SUBAPPLICATION Uebung_213c (* Standard IEC 61131-3 FB_CTU_UDINT (Vorwärtszähler, UDINT) mit Terminal-Ausgabe (PHYS_LREAL) *)
  (* Standard: 61131-3; Description: Copyright (c) 2026 Meisterschulen am Ostbahnhof This program and the accompanying materials are made available under the terms of the Eclipse Public License 2.0 which is available at https://www.eclipse.org/legal/epl-2.0/ SPDX-License-Identifier: EPL-2.0 *)
  (* Version 1.1, 2026-04-21, Franz Höpfinger, Meisterschulen am Ostbahnhof, Added terminal output for counter value (PHYS_LREAL, direct connection) *)
  (* Version 1.0, 2026-04-20, Franz Höpfinger, Meisterschulen am Ostbahnhof, initial API and implementation (IEC 61131-3 version) *)
  PACKAGE Uebungen;
  IMPORT Uebungen::const::UT::Horse::DefaultPool_Horse::Container_Horse;
  IMPORT Uebungen::const::UT::Horse::DefaultPool_Horse::ObjectPointer_Horse;
  IMPORT Uebungen::const::UT::Horse::DefaultPool_Horse::frame_00;
  IMPORT Uebungen::const::UT::Horse::DefaultPool_Horse::frame_01;
  IMPORT Uebungen::const::UT::Horse::DefaultPool_Horse::frame_02;
  IMPORT Uebungen::const::UT::Horse::DefaultPool_Horse::frame_03;
  IMPORT Uebungen::const::UT::Horse::DefaultPool_Horse::frame_04;
  IMPORT Uebungen::const::UT::Horse::DefaultPool_Horse::frame_05;
  IMPORT Uebungen::const::UT::Horse::DefaultPool_Horse::frame_06;
  IMPORT Uebungen::const::UT::Horse::DefaultPool_Horse::frame_07;
  IMPORT Uebungen::const::UT::Horse::DefaultPool_Horse::frame_08;
  IMPORT Uebungen::const::UT::Horse::DefaultPool_Horse::frame_09;
  IMPORT Uebungen::const::UT::Horse::DefaultPool_Horse::frame_10;
  IMPORT Uebungen::const::UT::Horse::DefaultPool_Horse::frame_11;
  IMPORT Uebungen::const::UT::Horse::DefaultPool_Horse::frame_12;
  IMPORT Uebungen::const::UT::Horse::DefaultPool_Horse::frame_13;
  IMPORT Uebungen::const::UT::Horse::DefaultPool_Horse::frame_14;
  IMPORT Uebungen::const::UT::Horse::DefaultPool_Horse::frame_15;
  IMPORT Uebungen::const::UT::Horse::DefaultPool_Horse::frame_16;
  IMPORT Uebungen::const::UT::Horse::DefaultPool_Horse::frame_17;
  IMPORT Uebungen::const::UT::Horse::DefaultPool_Horse::frame_18;
  IMPORT Uebungen::const::UT::Horse::DefaultPool_Horse::frame_19;
  IMPORT Uebungen::const::UT::Horse::DefaultPool_Horse::frame_20;
  IMPORT Uebungen::const::UT::Horse::DefaultPool_Horse::frame_21;
  IMPORT Uebungen::const::UT::Horse::DefaultPool_Horse::frame_22;
  IMPORT Uebungen::const::UT::Horse::DefaultPool_Horse::frame_23;
  IMPORT Uebungen::const::UT::Horse::DefaultPool_Horse::frame_24;
  IMPORT Uebungen::const::UT::Horse::DefaultPool_Horse::frame_25;
  IMPORT Uebungen::const::UT::Horse::DefaultPool_Horse::frame_26;
  IMPORT Uebungen::const::UT::Horse::DefaultPool_Horse::frame_27;
  IMPORT Uebungen::const::UT::Horse::DefaultPool_Horse::frame_28;
  IMPORT Uebungen::const::UT::Horse::DefaultPool_Horse::frame_29;
  IMPORT Uebungen::const::UT::Horse::DefaultPool_Horse::frame_30;
  IMPORT Uebungen::const::UT::Horse::DefaultPool_Horse::frame_31;
  IMPORT logiBUS::io::DI::logiBUS_DI::Input_I1;
  IMPORT logiBUS::io::DI::logiBUS_DI::Input_I2;
  IMPORT logiBUS::io::DI::logiBUS_DI_Events::BUTTON_SINGLE_CLICK;
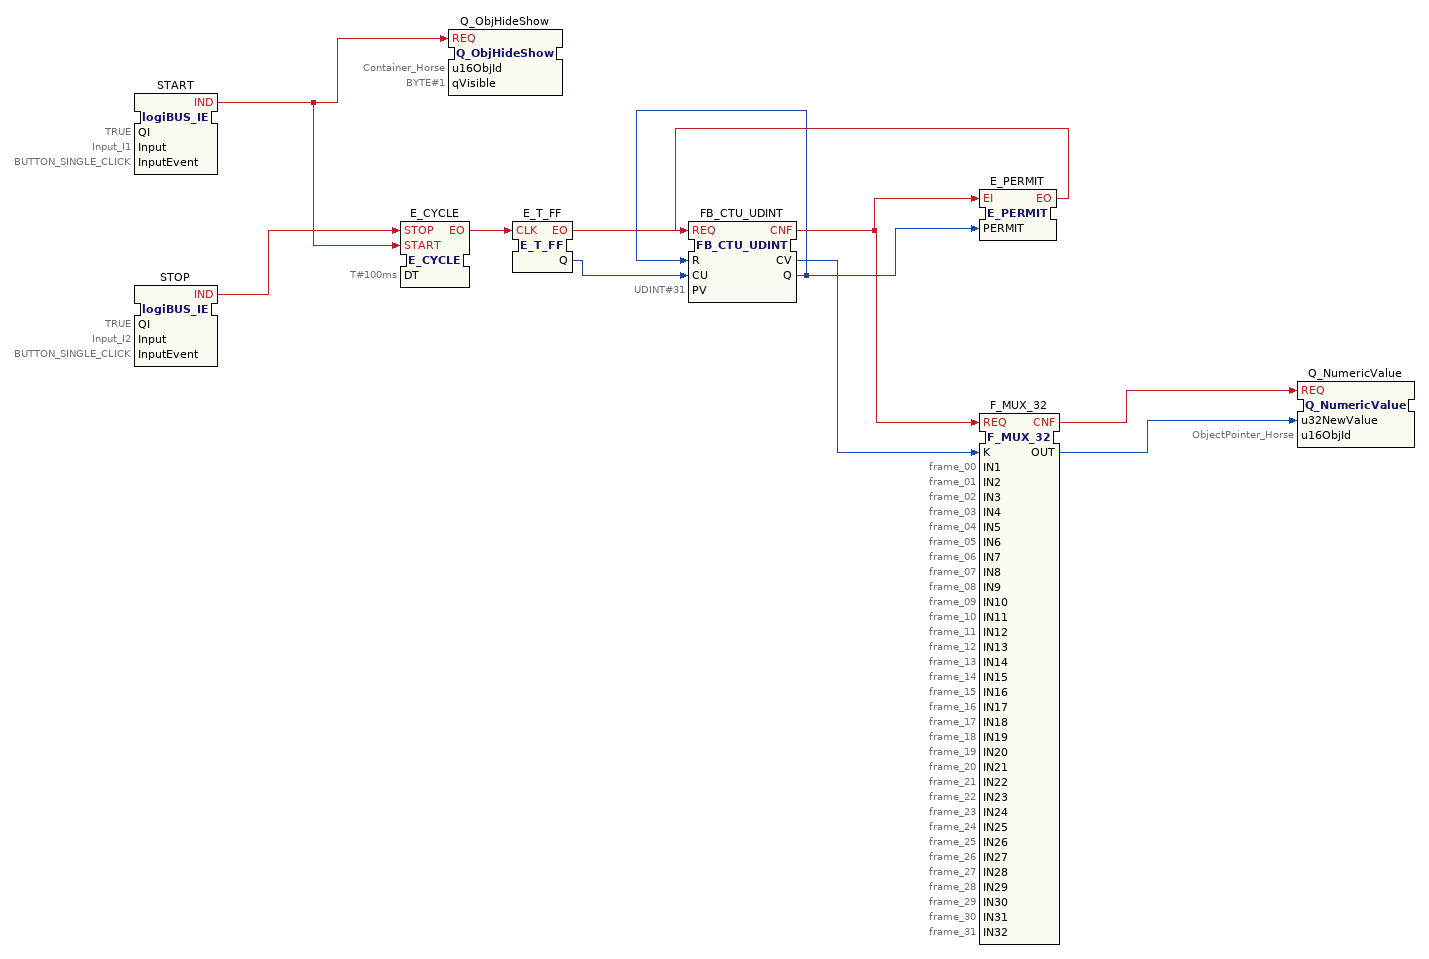
  FBS
    FB_CTU_UDINT : iec61131::counters::FB_CTU_UDINT(PV := UDINT#31);
    START : logiBUS::io::DI::logiBUS_IE(QI := TRUE, Input := Input_I1, InputEvent := BUTTON_SINGLE_CLICK);
    Q_NumericValue : isobus::UT::Q::Q_NumericValue(u16ObjId := ObjectPointer_Horse);
    F_MUX_32 : iec61131::selection::F_MUX_32(IN1 := frame_00, IN2 := frame_01, IN3 := frame_02, IN4 := frame_03, IN5 := frame_04, IN6 := frame_05, IN7 := frame_06, IN8 := frame_07, IN9 := frame_08, IN10 := frame_09, IN11 := frame_10, IN12 := frame_11, IN13 := frame_12, IN14 := frame_13, IN15 := frame_14, IN16 := frame_15, IN17 := frame_16, IN18 := frame_17, IN19 := frame_18, IN20 := frame_19, IN21 := frame_20, IN22 := frame_21, IN23 := frame_22, IN24 := frame_23, IN25 := frame_24, IN26 := frame_25, IN27 := frame_26, IN28 := frame_27, IN29 := frame_28, IN30 := frame_29, IN31 := frame_30, IN32 := frame_31);
    E_PERMIT : iec61499::events::E_PERMIT;
    E_CYCLE : iec61499::events::E_CYCLE(DT := T#100ms);
    STOP : logiBUS::io::DI::logiBUS_IE(QI := TRUE, Input := Input_I2, InputEvent := BUTTON_SINGLE_CLICK);
    E_T_FF : iec61499::events::E_T_FF;
    Q_ObjHideShow : isobus::UT::Q::Q_ObjHideShow(u16ObjId := Container_Horse, qVisible := BYTE#1);
  END_FBS
  EVENT_CONNECTIONS
    FB_CTU_UDINT.CNF TO F_MUX_32.REQ;
    F_MUX_32.CNF TO Q_NumericValue.REQ;
    FB_CTU_UDINT.CNF TO E_PERMIT.EI;
    E_PERMIT.EO TO FB_CTU_UDINT.REQ;
    STOP.IND TO E_CYCLE.STOP;
    E_CYCLE.EO TO E_T_FF.CLK;
    E_T_FF.EO TO FB_CTU_UDINT.REQ;
    START.IND TO E_CYCLE.START;
    START.IND TO Q_ObjHideShow.REQ;
  END_CONNECTIONS
  DATA_CONNECTIONS
    FB_CTU_UDINT.CV TO F_MUX_32.K;
    F_MUX_32.OUT TO Q_NumericValue.u32NewValue;
    FB_CTU_UDINT.Q TO FB_CTU_UDINT.R;
    FB_CTU_UDINT.Q TO E_PERMIT.PERMIT;
    E_T_FF.Q TO FB_CTU_UDINT.CU;
  END_CONNECTIONS
END_SUBAPPLICATION
